// LS Electric XG5000 project: 0122 PLC 데이터
// PLC LSPLC

PROGRAM NewProgram (task: 스캔 프로그램)

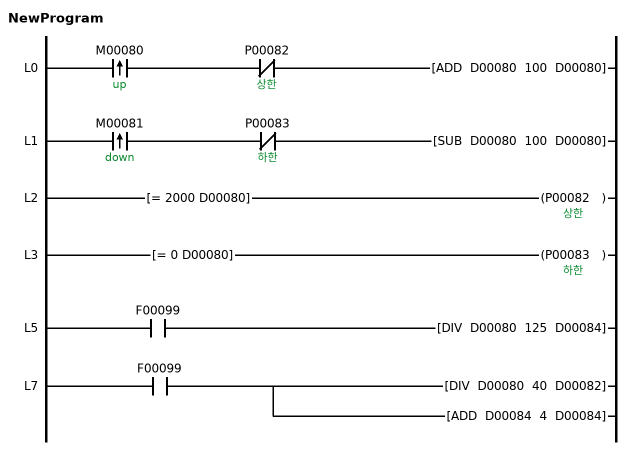
; L0
LOADP     M00080	// up
AND NOT   P00082	// 상한
ADD       D00080 100 D00080
; L1
LOADP     M00081	// down
AND NOT   P00083	// 하한
SUB       D00080 100 D00080
; L2
LOAD=     2000 D00080
OUT       P00082	// 상한
; L3
LOAD=     0 D00080
OUT       P00083	// 하한
; L5
LOAD      F00099
DIV       D00080 125 D00084
; L7
LOAD      F00099
DIV       D00080 40 D00082
ADD       D00084 4 D00084

VARIABLES AND COMMENTS (devices not used above)
M00010	BIT	스위치 1
D00000	WORD	전번
M00001	BIT	스위치2
D00022	WORD	현재카운터수
M00002	BIT	스위치3
M00003	BIT	카운터
M00004	BIT	카운터 리셋
C0000	BIT/WORD	카운트
M00000	BIT	스위치1
P00081	BIT	하한